{attribute 'qualified_only'}
VAR_GLOBAL
END_VAR

(* stored: Version 1.1.0.1, ProductVersion 3.1.4024.10
   GVL P_Sensors: Id {e60c22bd-67fb-4985-bb27-7274310d52c7} *)
